{attribute 'OPC.UA.DA.StructuredType' := '1'}
FUNCTION_BLOCK FB_BaseMachine
VAR

	{attribute 'OPC.UA.DA' := '0'} 
	bBusy: BOOL := FALSE;
	{attribute 'OPC.UA.DA' := '1'} 
	bError: BOOL := FALSE;
	{attribute 'OPC.UA.DA' := '1'} 
	bEnable: BOOL := FALSE;
	{attribute 'OPC.UA.DA' := '1'} 
	eState: E_MachineState := E_MachineState.IDLE;
	{attribute 'OPC.UA.DA' := '1'} 
	{attribute 'OPC.UA.DA.StructuredType' := '1'}
	fbSequenceManager: FB_SequenceManager;
	{attribute 'OPC.UA.DA' := '0'} 
	aAllComponents: ARRAY[1..50] OF POINTER TO FB_BaseDevice;
	
	{attribute 'OPC.UA.DA' := '1'} 
	aErrors: ARRAY[1..20] OF ST_Alarm;	// raiseEvent() method updates Error1 / aErrors[1] only at the moment, must implement a ring buffer with error active checking for full functionality

	
END_VAR 

VAR_INPUT
	{attribute 'OPC.UA.DA' := '1'} 
	sID: STRING;  
	{attribute 'OPC.UA.DA' := '1'} 
	sDescr: STRING;
	{attribute 'OPC.UA.DA' := '1'} 
	nQtyComponents: INT;
END_VAR

METHOD devices_disable_All : BOOL
VAR
	iterator: INT;
	
END_VAR
FOR iterator:=1 TO nQtyComponents BY 1 DO
	aAllComponents[iterator]^.disable();
END_FOR
END_METHOD

METHOD devices_disable_CurrSeq : BOOL
VAR
	iterator: INT;
	Steps : ARRAY[1..20] OF ST_SequenceStep;
END_VAR
FOR iterator:=1 TO fbSequenceManager.getCurrentSeq_FB()^.stepsTotal() BY 1 DO
	
	Steps := fbSequenceManager.getCurrentSeq_FB()^.steps();
	Steps[iterator].Device^.disable();
	
END_FOR
END_METHOD

METHOD devices_enable_All : BOOL
VAR
	iterator: INT;
END_VAR
FOR iterator:=1 TO nQtyComponents BY 1 DO
	aAllComponents[iterator]^.enable();
END_FOR
END_METHOD

METHOD devices_enable_CurrSeq : BOOL
VAR
	iterator: INT;
	Steps : ARRAY[1..20] OF ST_SequenceStep;
END_VAR
FOR iterator:=1 TO fbSequenceManager.getCurrentSeq_FB()^.stepsTotal() BY 1 DO
	Steps := fbSequenceManager.getCurrentSeq_FB()^.steps();
	Steps[iterator].Device^.enable();
END_FOR
END_METHOD

METHOD devices_setAuto_All : BOOL
VAR
	iterator: INT;
END_VAR
FOR iterator:=1 TO nQtyComponents BY 1 DO
	aAllComponents[iterator]^.setMode(Mode := E_DeviceMode.AUTO);
END_FOR
END_METHOD

METHOD devices_setAuto_CurrSeq : BOOL
VAR
	iterator: INT;
	Steps : ARRAY[1..20] OF ST_SequenceStep;
END_VAR
FOR iterator:=1 TO fbSequenceManager.getCurrentSeq_FB()^.stepsTotal() BY 1 DO
	
	Steps := fbSequenceManager.getCurrentSeq_FB()^.steps();
	Steps[iterator].Device^.setMode(Mode := E_DeviceMode.AUTO);
END_FOR
END_METHOD

METHOD devices_setManual_All : BOOL
VAR
	iterator: INT;
END_VAR
FOR iterator:=1 TO nQtyComponents BY 1 DO
	aAllComponents[iterator]^.setMode(Mode := E_DeviceMode.AUTO);
END_FOR
END_METHOD

METHOD devices_setManual_CurrSeq : BOOL
VAR
	iterator: INT;
	Steps : ARRAY[1..20] OF ST_SequenceStep;
END_VAR
FOR iterator:=1 TO fbSequenceManager.getCurrentSeq_FB()^.stepsTotal() BY 1 DO
	
	Steps := fbSequenceManager.getCurrentSeq_FB()^.steps();
	Steps[iterator].Device^.setMode(Mode := E_DeviceMode.MANUAL);
END_FOR
END_METHOD

METHOD seq_Pause : BOOL
VAR_INPUT
END_VAR
fbSequenceManager.pauseSequence();
END_METHOD

METHOD seq_Start : BOOL
VAR_INPUT
	SeqNum: UINT;
END_VAR
devices_disable_All();
fbSequenceManager.selectSequence(Sequence := 1);
devices_enable_CurrSeq();
fbSequenceManager.startSequence();
END_METHOD

METHOD seq_Stop : BOOL
VAR_INPUT
END_VAR
fbSequenceManager.stopSequence();
END_METHOD

END_FUNCTION_BLOCK

(* stored: Version 1.1.0.1, ProductVersion 3.1.4024.12
   POU FB_BaseMachine: Id {6ab281f6-25bb-4cb2-98da-8fb2f940b9cd}, SpecialFunc None
   Method devices_disable_All: Id {d244f351-60e3-4280-ab38-d2f479e80693}
   Method devices_disable_CurrSeq: Id {817dca39-f242-4aa7-9a18-de59e2831eb6}
   Method devices_enable_All: Id {2d5bb57e-f62f-4d54-9a86-b18d71deee3e}
   Method devices_enable_CurrSeq: Id {550e4379-d359-40ab-b762-42d88501c446}
   Method devices_setAuto_All: Id {44b6de1d-80f7-48b6-8b11-23cf806f7ffc}
   Method devices_setAuto_CurrSeq: Id {48a97b93-3542-44cf-932a-920144fa55a6}
   Method devices_setManual_All: Id {820e5822-0b50-4978-9aa1-512ccb6baa9c}
   Method devices_setManual_CurrSeq: Id {50e4b034-7cce-4db5-818c-7f74c9807537}
   Method seq_Pause: Id {dcf13c55-b5ac-44bd-9861-9f3985e52050}
   Method seq_Start: Id {16b9da48-2ae5-47cb-b10d-16db289d1f6e}
   Method seq_Stop: Id {b22b4d46-f25e-4eb7-a917-e47b5fc4aab8} *)
